{attribute 'OPC.UA.DA' := '1'}    
TYPE ST_AO :
STRUCT
		Value		  AT %Q*	: INT	;
		Description 			: STRING	;

END_STRUCT
END_TYPE

(* stored: Version 1.1.0.1, ProductVersion 3.1.4024.12
   DUT ST_AO: Id {afbf683e-d623-4191-a01d-e0767348f253} *)
